(* Logix 5000 project; controller L3 vendor 1 type 14 code 92 rev 20.12; software revision 20.04; part 4 of 9 *)
(* tags used below, declared in another part *)
   B3 : DINT[100];
   L3_stat : DINT[20];
   N20 : DINT[200];
   N21 : DINT[200];
   N7 : DINT[200];
   N9 : DINT[200];   // niveau decapage vers lancy (n9[10) ;;N9[70]
   NCOM : INT[20];
   new_def_decap : BOOL;
   s_def_new : DINT;
   s_def_old : DINT;
   stat_L3 : DINT[20];
   T4 : TIMER[180];
(* _2_GENERAL, continued *)

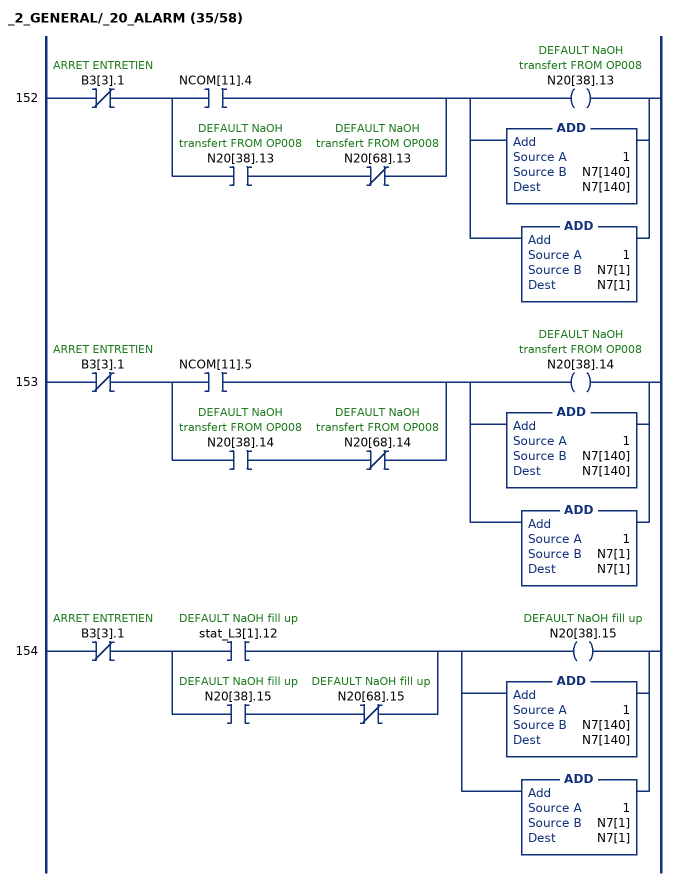
   [picture p50: _2_GENERAL/_20_ALARM rungs 152-154]
   152: XIO(B3[3].1)[XIC(NCOM[11].4) ,XIC(N20[38].13) XIO(N20[68].13) ][OTE(N20[38].13) ,ADD(1,N7[140],N7[140]) ,ADD(1,N7[1],N7[1]) ];
   153: XIO(B3[3].1)[XIC(NCOM[11].5) ,XIC(N20[38].14) XIO(N20[68].14) ][OTE(N20[38].14) ,ADD(1,N7[140],N7[140]) ,ADD(1,N7[1],N7[1]) ];
   154: XIO(B3[3].1)[XIC(stat_L3[1].12) ,XIC(N20[38].15) XIO(N20[68].15) ][OTE(N20[38].15) ,ADD(1,N7[140],N7[140]) ,ADD(1,N7[1],N7[1]) ];
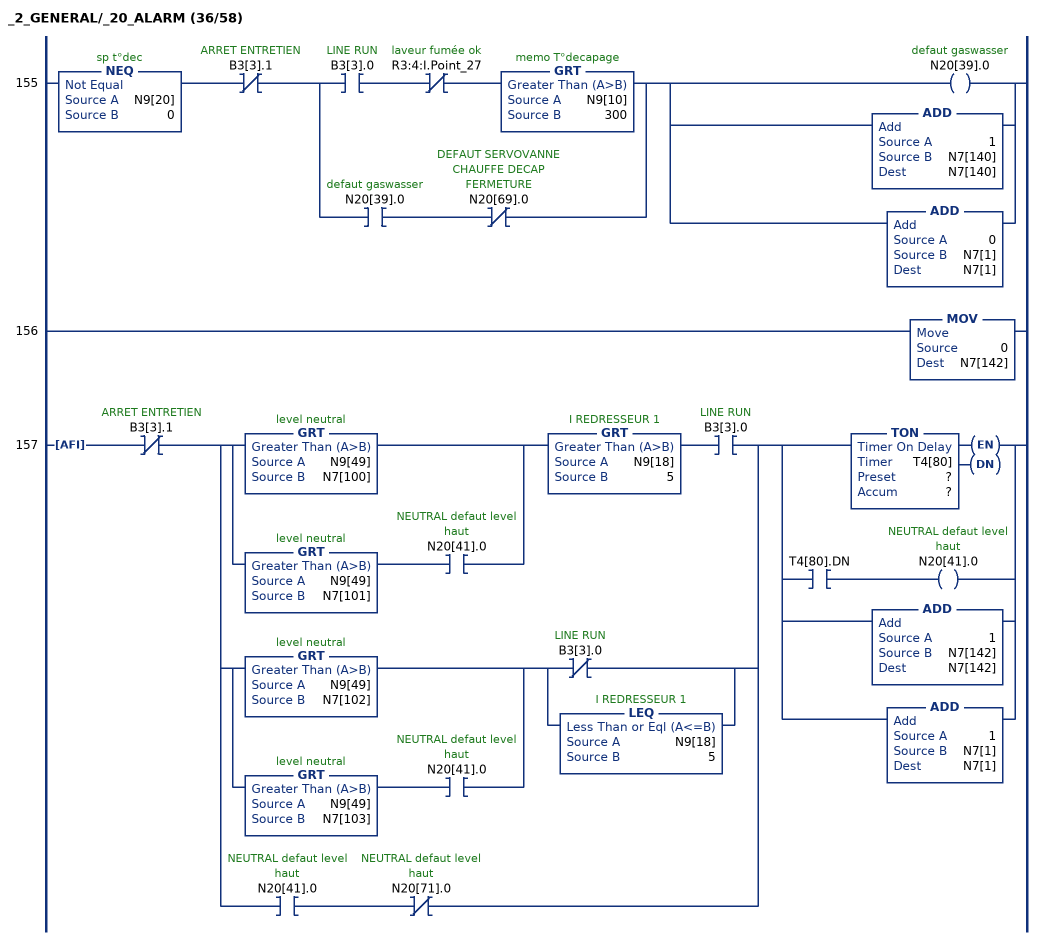
   155: NEQ(N9[20],0)XIO(B3[3].1)[XIC(B3[3].0) XIO(R3:4:I.Point_27) GRT(N9[10],300) ,XIC(N20[39].0) XIO(N20[69].0) ][OTE(N20[39].0) ,ADD(1,N7[140],N7[140]) ,ADD(0,N7[1],N7[1]) ];
   156: MOV(0,N7[142]);
   157: AFI()XIO(B3[3].1)[[GRT(N9[49],N7[100]) ,GRT(N9[49],N7[101]) XIC(N20[41].0) ] GRT(N9[18],5) XIC(B3[3].0) ,[GRT(N9[49],N7[102]) ,GRT(N9[49],N7[103]) XIC(N20[41].0) ] [XIO(B3[3].0) ,LEQ(N9[18],5) ] ,XIC(N20[41].0) XIO(N20[71].0) ][TON(T4[80],?,?) ,XIC(T4[80].DN) OTE(N20[41].0) ,ADD(1,N7[142],N7[142]) ,ADD(1,N7[1],N7[1]) ];
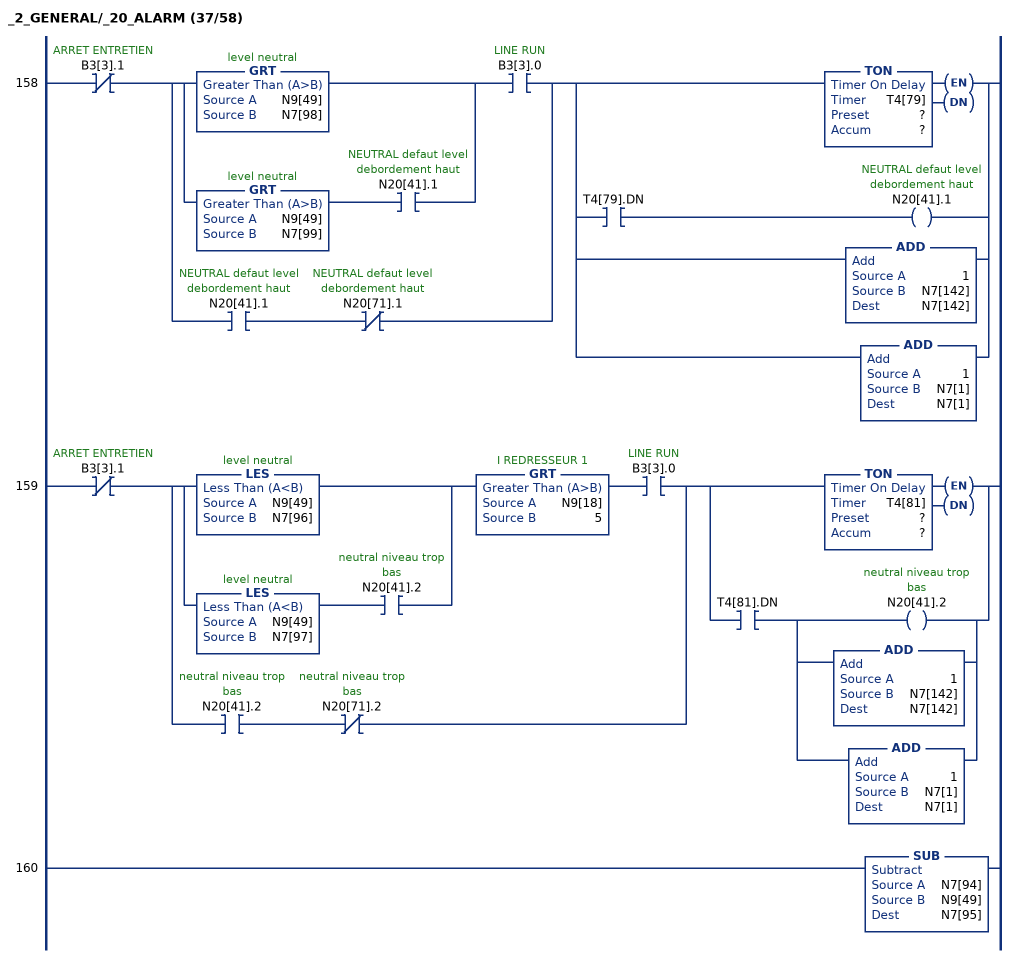
   158: XIO(B3[3].1)[[GRT(N9[49],N7[98]) ,GRT(N9[49],N7[99]) XIC(N20[41].1) ] XIC(B3[3].0) ,XIC(N20[41].1) XIO(N20[71].1) ][TON(T4[79],?,?) ,XIC(T4[79].DN) OTE(N20[41].1) ,ADD(1,N7[142],N7[142]) ,ADD(1,N7[1],N7[1]) ];
   159: XIO(B3[3].1)[[LES(N9[49],N7[96]) ,LES(N9[49],N7[97]) XIC(N20[41].2) ] GRT(N9[18],5) XIC(B3[3].0) ,XIC(N20[41].2) XIO(N20[71].2) ][TON(T4[81],?,?) ,XIC(T4[81].DN) [OTE(N20[41].2) ,ADD(1,N7[142],N7[142]) ,ADD(1,N7[1],N7[1]) ] ];
   160: SUB(N7[94],N9[49],N7[95]);
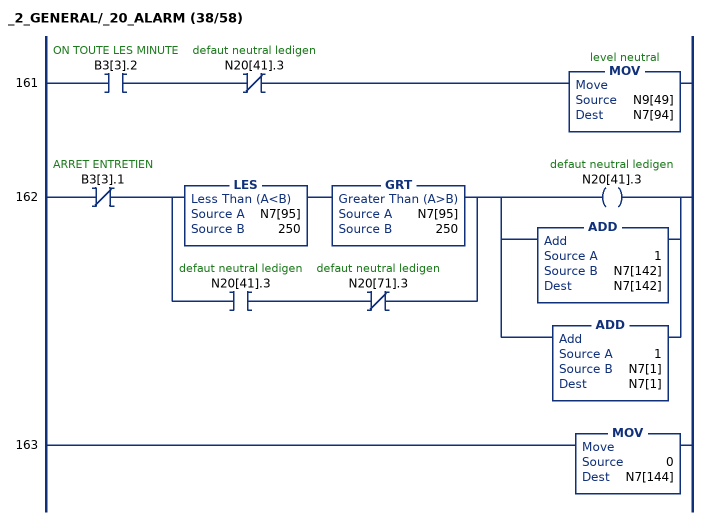
   161: XIC(B3[3].2)XIO(N20[41].3)MOV(N9[49],N7[94]);
   162: XIO(B3[3].1)[LES(N7[95],250) GRT(N7[95],250) ,XIC(N20[41].3) XIO(N20[71].3) ][OTE(N20[41].3) ,ADD(1,N7[142],N7[142]) ,ADD(1,N7[1],N7[1]) ];
   163: MOV(0,N7[144]);
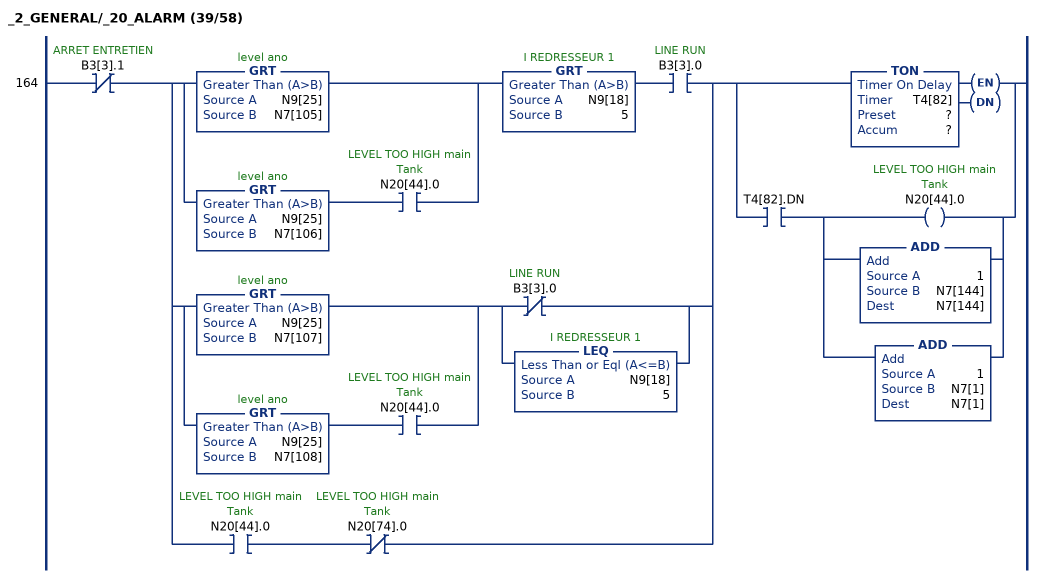
   164: XIO(B3[3].1)[[GRT(N9[25],N7[105]) ,GRT(N9[25],N7[106]) XIC(N20[44].0) ] GRT(N9[18],5) XIC(B3[3].0) ,[GRT(N9[25],N7[107]) ,GRT(N9[25],N7[108]) XIC(N20[44].0) ] [XIO(B3[3].0) ,LEQ(N9[18],5) ] ,XIC(N20[44].0) XIO(N20[74].0) ][TON(T4[82],?,?) ,XIC(T4[82].DN) [OTE(N20[44].0) ,ADD(1,N7[144],N7[144]) ,ADD(1,N7[1],N7[1]) ] ];
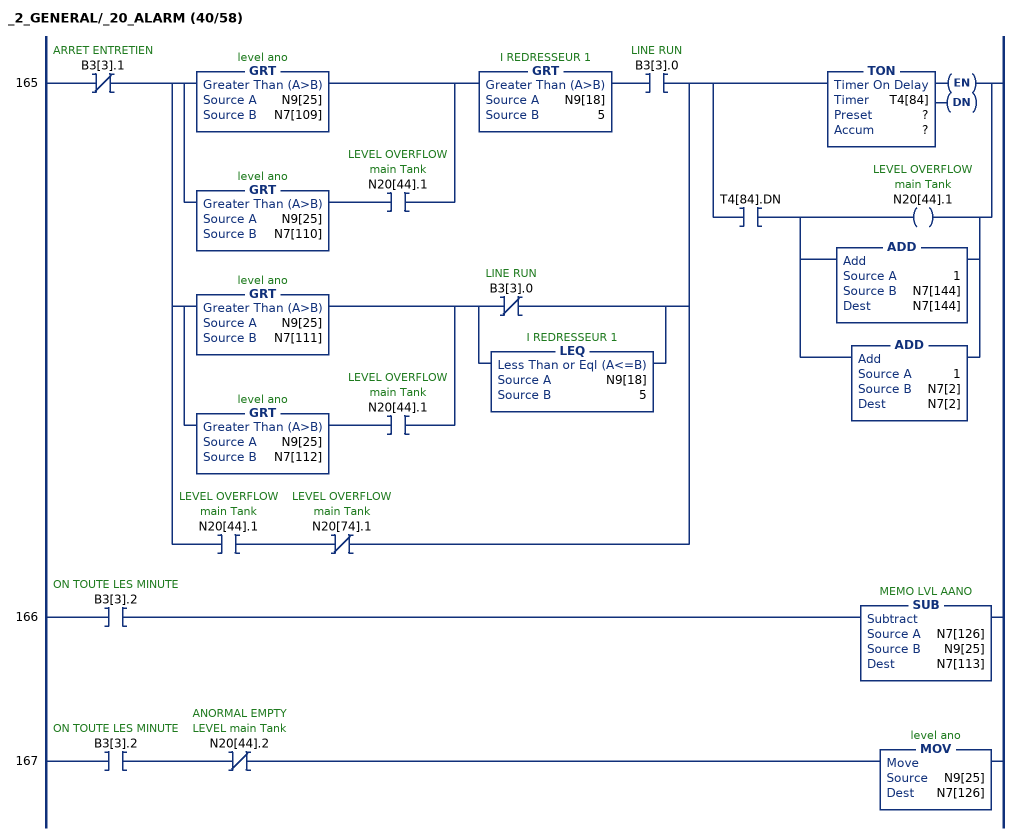
   165: XIO(B3[3].1)[[GRT(N9[25],N7[109]) ,GRT(N9[25],N7[110]) XIC(N20[44].1) ] GRT(N9[18],5) XIC(B3[3].0) ,[GRT(N9[25],N7[111]) ,GRT(N9[25],N7[112]) XIC(N20[44].1) ] [XIO(B3[3].0) ,LEQ(N9[18],5) ] ,XIC(N20[44].1) XIO(N20[74].1) ][TON(T4[84],?,?) ,XIC(T4[84].DN) [OTE(N20[44].1) ,ADD(1,N7[144],N7[144]) ,ADD(1,N7[2],N7[2]) ] ];
   166: XIC(B3[3].2)SUB(N7[126],N9[25],N7[113]);
   167: XIC(B3[3].2)XIO(N20[44].2)MOV(N9[25],N7[126]);
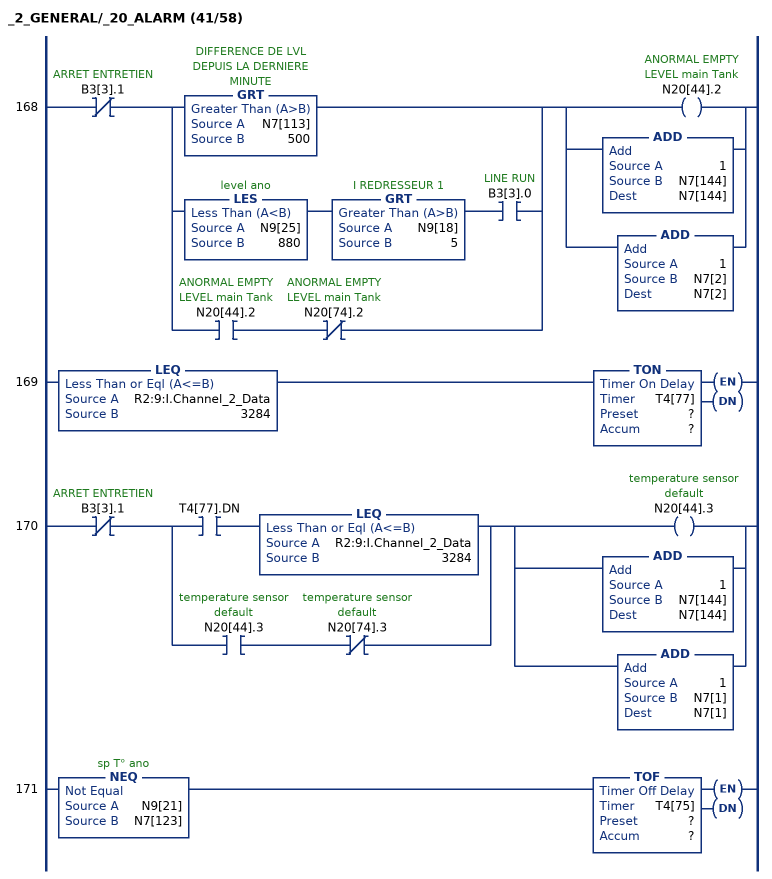
   168: XIO(B3[3].1)[GRT(N7[113],500) ,LES(N9[25],880) GRT(N9[18],5) XIC(B3[3].0) ,XIC(N20[44].2) XIO(N20[74].2) ][OTE(N20[44].2) ,ADD(1,N7[144],N7[144]) ,ADD(1,N7[2],N7[2]) ];
   169: LEQ(R2:9:I.Channel_2_Data,3284)TON(T4[77],?,?);
   170: XIO(B3[3].1)[XIC(T4[77].DN) LEQ(R2:9:I.Channel_2_Data,3284) ,XIC(N20[44].3) XIO(N20[74].3) ][OTE(N20[44].3) ,ADD(1,N7[144],N7[144]) ,ADD(1,N7[1],N7[1]) ];
   171: NEQ(N9[21],N7[123])TOF(T4[75],?,?);
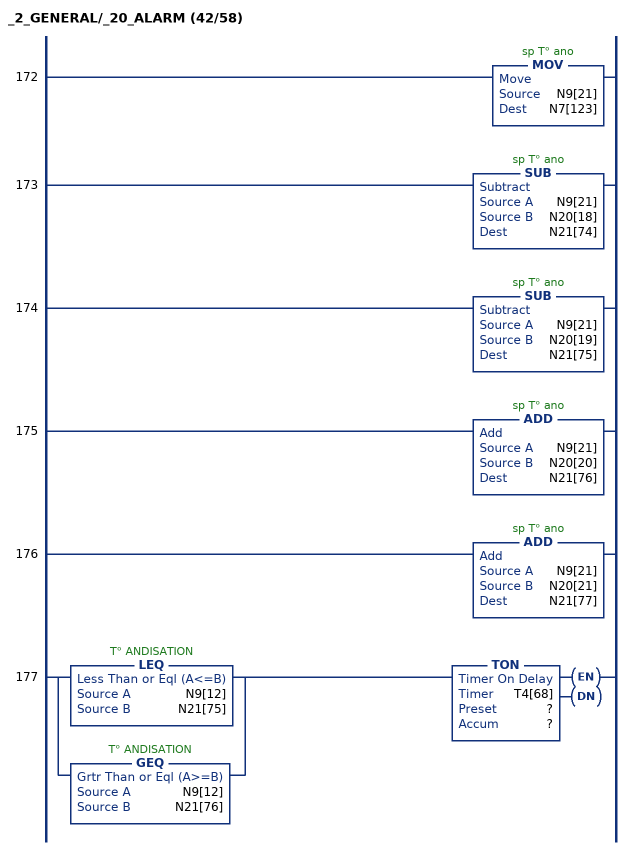
   172: MOV(N9[21],N7[123]);
   173: SUB(N9[21],N20[18],N21[74]);
   174: SUB(N9[21],N20[19],N21[75]);
   175: ADD(N9[21],N20[20],N21[76]);
   176: ADD(N9[21],N20[21],N21[77]);
   177: [LEQ(N9[12],N21[75]) ,GEQ(N9[12],N21[76]) ]TON(T4[68],?,?);
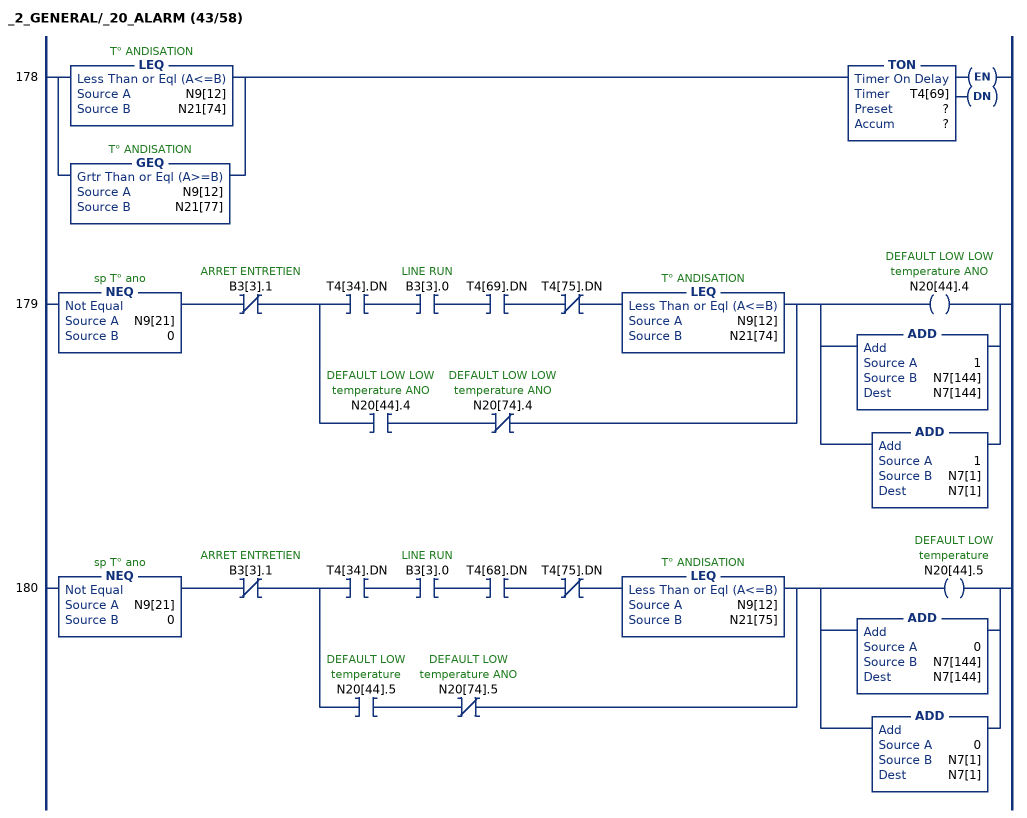
   178: [LEQ(N9[12],N21[74]) ,GEQ(N9[12],N21[77]) ]TON(T4[69],?,?);
   179: NEQ(N9[21],0)XIO(B3[3].1)[XIC(T4[34].DN) XIC(B3[3].0) XIC(T4[69].DN) XIO(T4[75].DN) LEQ(N9[12],N21[74]) ,XIC(N20[44].4) XIO(N20[74].4) ][OTE(N20[44].4) ,ADD(1,N7[144],N7[144]) ,ADD(1,N7[1],N7[1]) ];
   180: NEQ(N9[21],0)XIO(B3[3].1)[XIC(T4[34].DN) XIC(B3[3].0) XIC(T4[68].DN) XIO(T4[75].DN) LEQ(N9[12],N21[75]) ,XIC(N20[44].5) XIO(N20[74].5) ][OTE(N20[44].5) ,ADD(0,N7[144],N7[144]) ,ADD(0,N7[1],N7[1]) ];
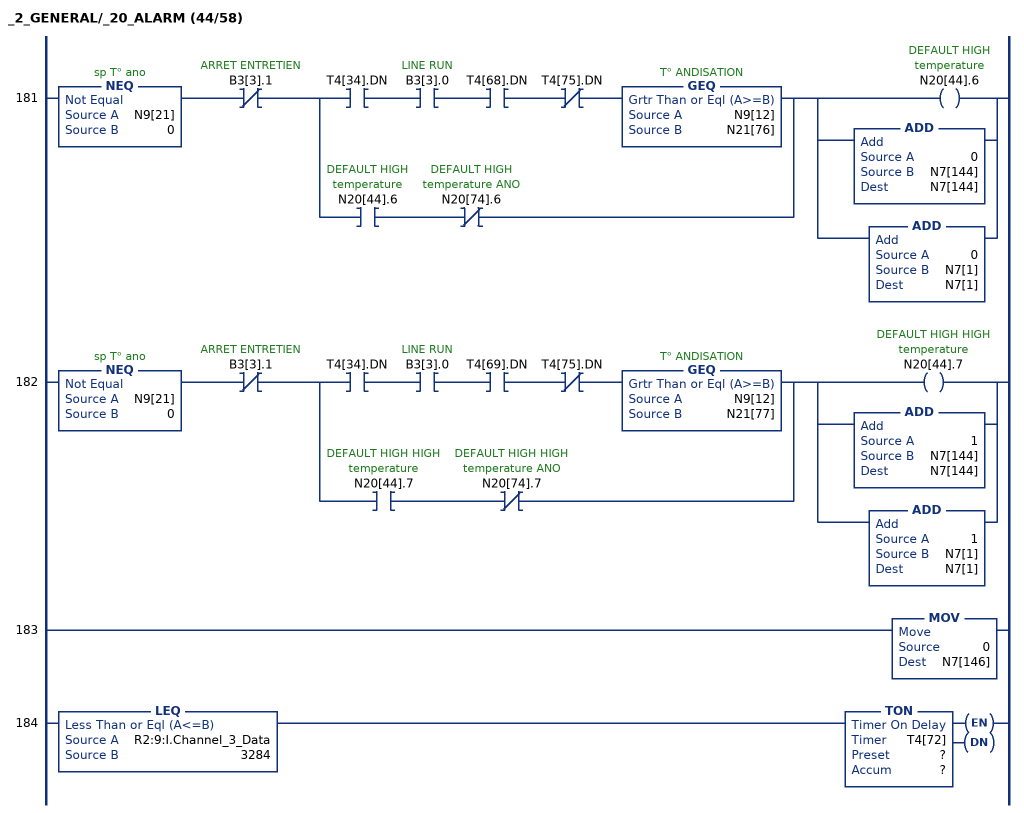
   181: NEQ(N9[21],0)XIO(B3[3].1)[XIC(T4[34].DN) XIC(B3[3].0) XIC(T4[68].DN) XIO(T4[75].DN) GEQ(N9[12],N21[76]) ,XIC(N20[44].6) XIO(N20[74].6) ][OTE(N20[44].6) ,ADD(0,N7[144],N7[144]) ,ADD(0,N7[1],N7[1]) ];
   182: NEQ(N9[21],0)XIO(B3[3].1)[XIC(T4[34].DN) XIC(B3[3].0) XIC(T4[69].DN) XIO(T4[75].DN) GEQ(N9[12],N21[77]) ,XIC(N20[44].7) XIO(N20[74].7) ][OTE(N20[44].7) ,ADD(1,N7[144],N7[144]) ,ADD(1,N7[1],N7[1]) ];
   183: MOV(0,N7[146]);
   184: LEQ(R2:9:I.Channel_3_Data,3284)TON(T4[72],?,?);
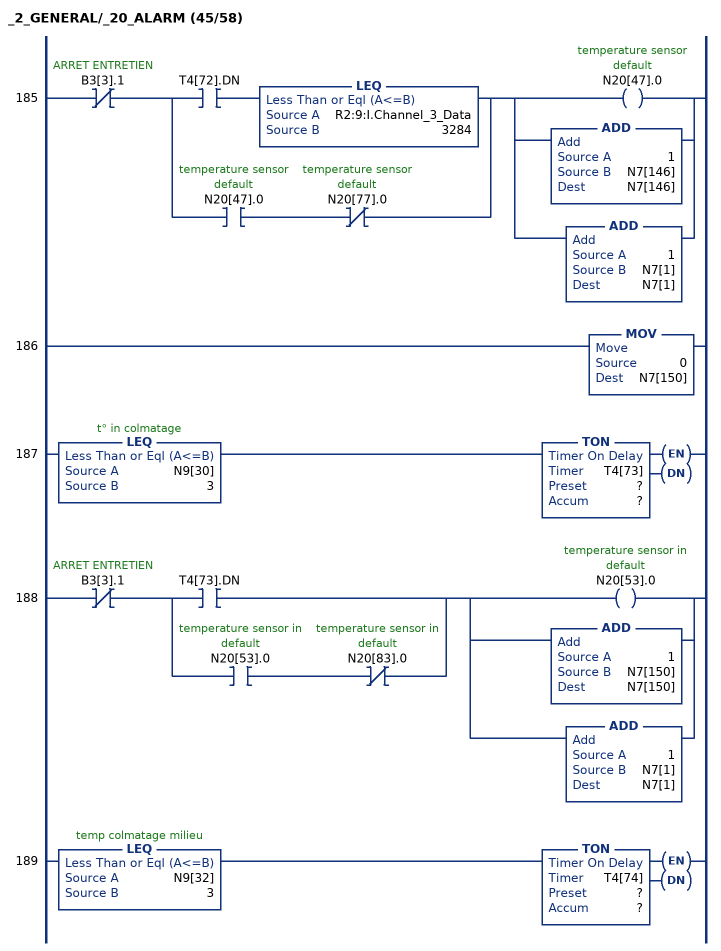
   185: XIO(B3[3].1)[XIC(T4[72].DN) LEQ(R2:9:I.Channel_3_Data,3284) ,XIC(N20[47].0) XIO(N20[77].0) ][OTE(N20[47].0) ,ADD(1,N7[146],N7[146]) ,ADD(1,N7[1],N7[1]) ];
   186: MOV(0,N7[150]);
   187: LEQ(N9[30],3)TON(T4[73],?,?);
   188: XIO(B3[3].1)[XIC(T4[73].DN) ,XIC(N20[53].0) XIO(N20[83].0) ][OTE(N20[53].0) ,ADD(1,N7[150],N7[150]) ,ADD(1,N7[1],N7[1]) ];
   189: LEQ(N9[32],3)TON(T4[74],?,?);
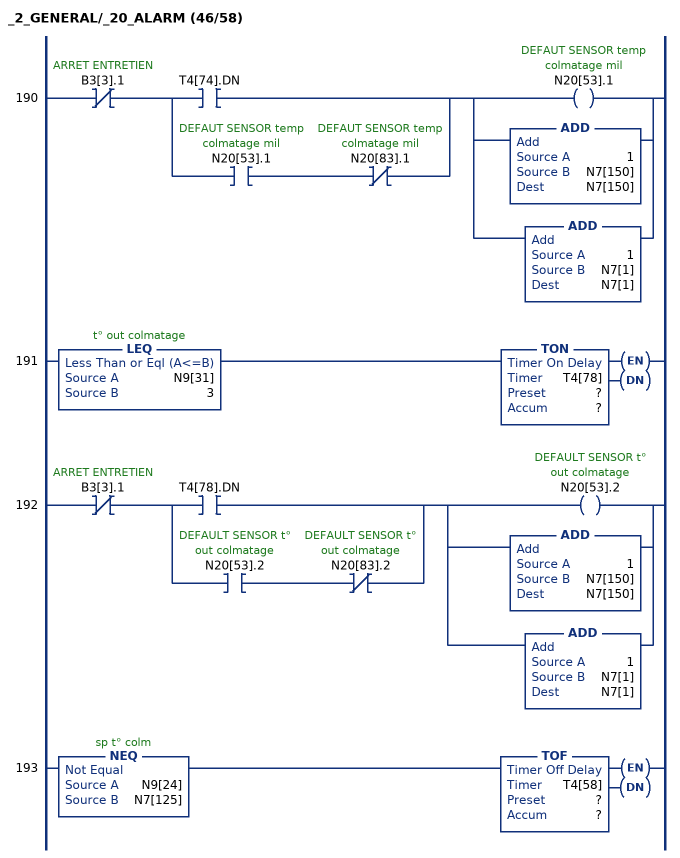
   190: XIO(B3[3].1)[XIC(T4[74].DN) ,XIC(N20[53].1) XIO(N20[83].1) ][OTE(N20[53].1) ,ADD(1,N7[150],N7[150]) ,ADD(1,N7[1],N7[1]) ];
   191: LEQ(N9[31],3)TON(T4[78],?,?);
   192: XIO(B3[3].1)[XIC(T4[78].DN) ,XIC(N20[53].2) XIO(N20[83].2) ][OTE(N20[53].2) ,ADD(1,N7[150],N7[150]) ,ADD(1,N7[1],N7[1]) ];
   193: NEQ(N9[24],N7[125])TOF(T4[58],?,?);
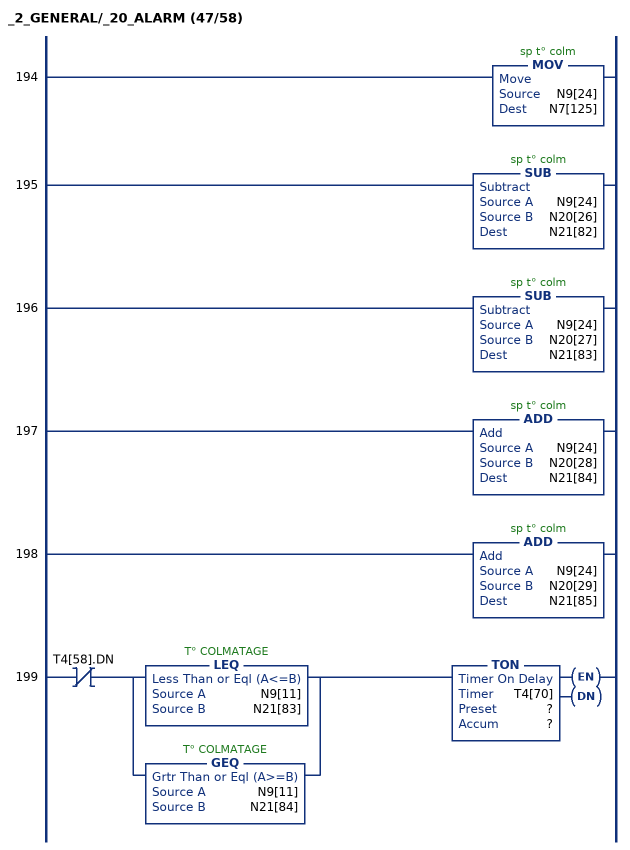
   194: MOV(N9[24],N7[125]);
   195: SUB(N9[24],N20[26],N21[82]);
   196: SUB(N9[24],N20[27],N21[83]);
   197: ADD(N9[24],N20[28],N21[84]);
   198: ADD(N9[24],N20[29],N21[85]);
   199: XIO(T4[58].DN)[LEQ(N9[11],N21[83]) ,GEQ(N9[11],N21[84]) ]TON(T4[70],?,?);
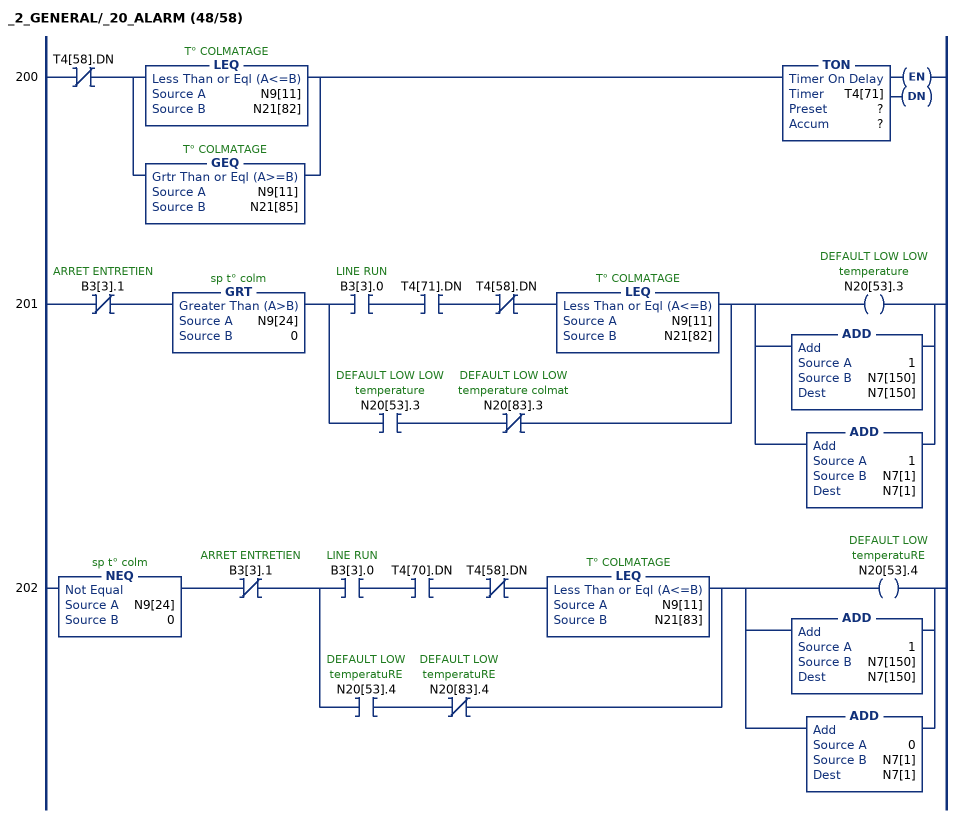
   200: XIO(T4[58].DN)[LEQ(N9[11],N21[82]) ,GEQ(N9[11],N21[85]) ]TON(T4[71],?,?);
   201: XIO(B3[3].1)GRT(N9[24],0)[XIC(B3[3].0) XIC(T4[71].DN) XIO(T4[58].DN) LEQ(N9[11],N21[82]) ,XIC(N20[53].3) XIO(N20[83].3) ][OTE(N20[53].3) ,ADD(1,N7[150],N7[150]) ,ADD(1,N7[1],N7[1]) ];
   202: NEQ(N9[24],0)XIO(B3[3].1)[XIC(B3[3].0) XIC(T4[70].DN) XIO(T4[58].DN) LEQ(N9[11],N21[83]) ,XIC(N20[53].4) XIO(N20[83].4) ][OTE(N20[53].4) ,ADD(1,N7[150],N7[150]) ,ADD(0,N7[1],N7[1]) ];
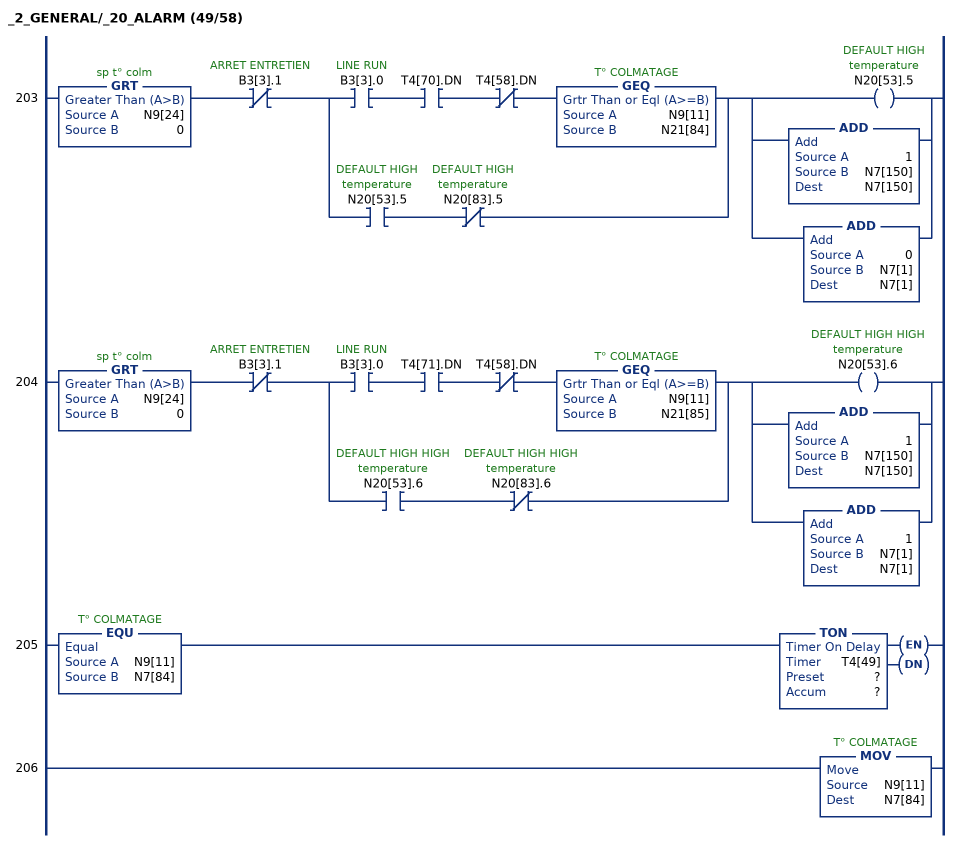
   203: GRT(N9[24],0)XIO(B3[3].1)[XIC(B3[3].0) XIC(T4[70].DN) XIO(T4[58].DN) GEQ(N9[11],N21[84]) ,XIC(N20[53].5) XIO(N20[83].5) ][OTE(N20[53].5) ,ADD(1,N7[150],N7[150]) ,ADD(0,N7[1],N7[1]) ];
   204: GRT(N9[24],0)XIO(B3[3].1)[XIC(B3[3].0) XIC(T4[71].DN) XIO(T4[58].DN) GEQ(N9[11],N21[85]) ,XIC(N20[53].6) XIO(N20[83].6) ][OTE(N20[53].6) ,ADD(1,N7[150],N7[150]) ,ADD(1,N7[1],N7[1]) ];
   205: EQU(N9[11],N7[84])TON(T4[49],?,?);
   206: MOV(N9[11],N7[84]);
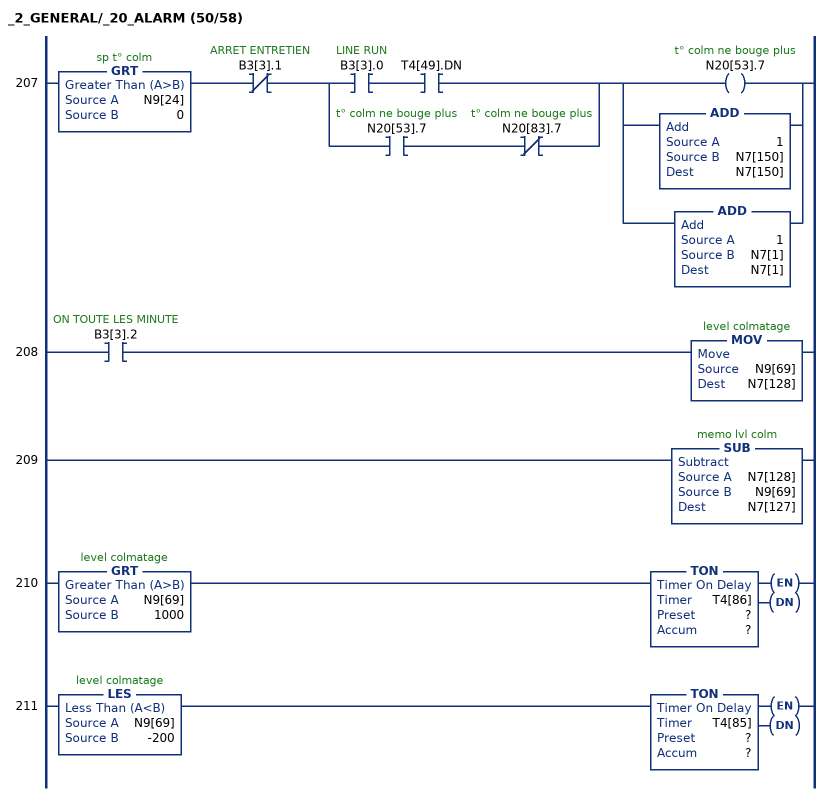
   207: GRT(N9[24],0)XIO(B3[3].1)[XIC(B3[3].0) XIC(T4[49].DN) ,XIC(N20[53].7) XIO(N20[83].7) ][OTE(N20[53].7) ,ADD(1,N7[150],N7[150]) ,ADD(1,N7[1],N7[1]) ];
   208: XIC(B3[3].2)MOV(N9[69],N7[128]);
   209: SUB(N7[128],N9[69],N7[127]);
   210: GRT(N9[69],1000)TON(T4[86],?,?);
   211: LES(N9[69],-200)TON(T4[85],?,?);
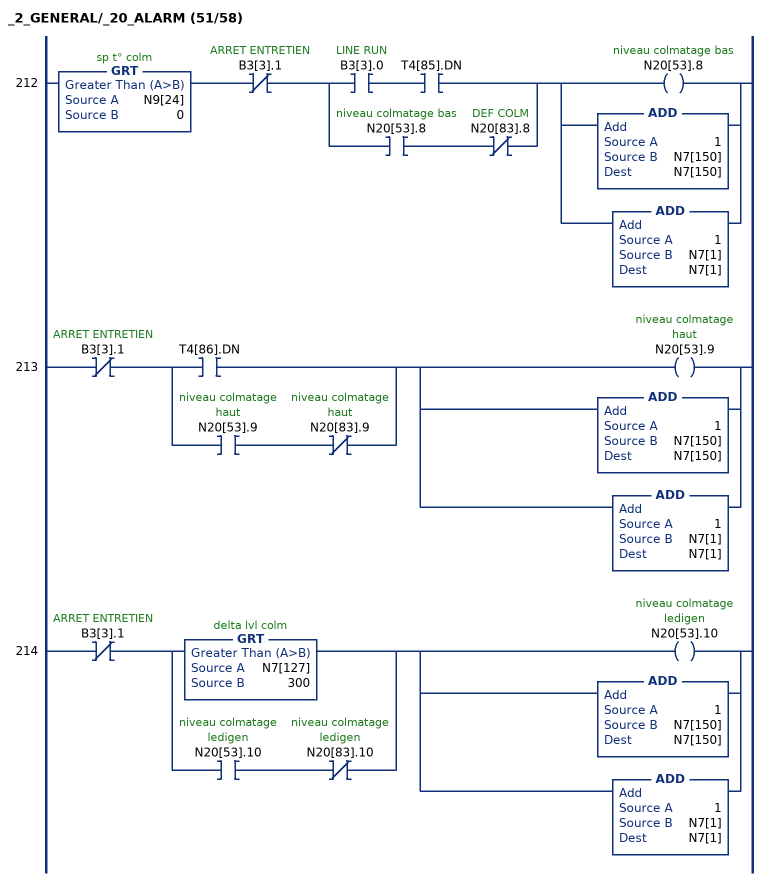
   212: GRT(N9[24],0)XIO(B3[3].1)[XIC(B3[3].0) XIC(T4[85].DN) ,XIC(N20[53].8) XIO(N20[83].8) ][OTE(N20[53].8) ,ADD(1,N7[150],N7[150]) ,ADD(1,N7[1],N7[1]) ];
   213: XIO(B3[3].1)[XIC(T4[86].DN) ,XIC(N20[53].9) XIO(N20[83].9) ][OTE(N20[53].9) ,ADD(1,N7[150],N7[150]) ,ADD(1,N7[1],N7[1]) ];
   214: XIO(B3[3].1)[GRT(N7[127],300) ,XIC(N20[53].10) XIO(N20[83].10) ][OTE(N20[53].10) ,ADD(1,N7[150],N7[150]) ,ADD(1,N7[1],N7[1]) ];
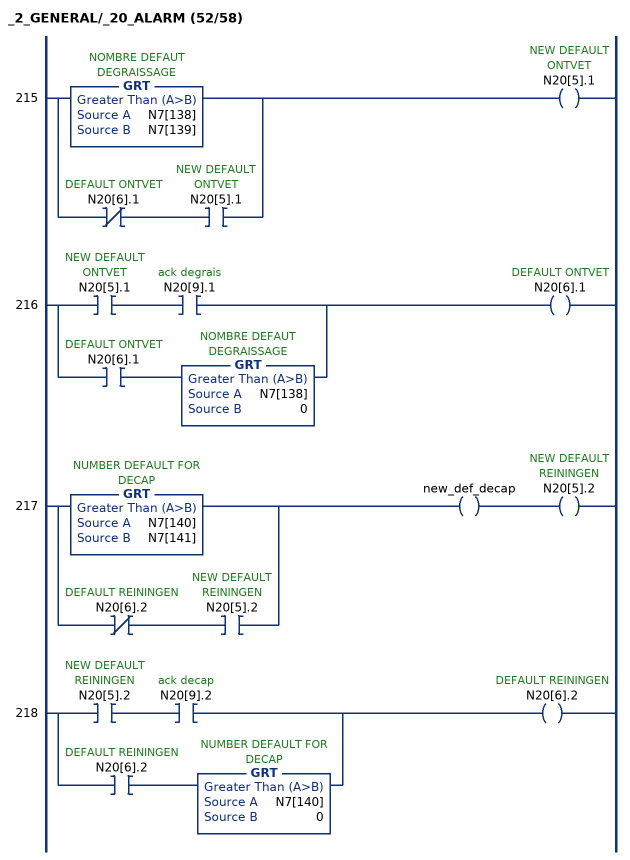
   215: [GRT(N7[138],N7[139]) ,XIO(N20[6].1) XIC(N20[5].1) ]OTE(N20[5].1);
   216: [XIC(N20[5].1) XIC(N20[9].1) ,XIC(N20[6].1) GRT(N7[138],0) ]OTE(N20[6].1);
   217: [GRT(N7[140],N7[141]) ,XIO(N20[6].2) XIC(N20[5].2) ]OTE(new_def_decap)OTE(N20[5].2);
   218: [XIC(N20[5].2) XIC(N20[9].2) ,XIC(N20[6].2) GRT(N7[140],0) ]OTE(N20[6].2);
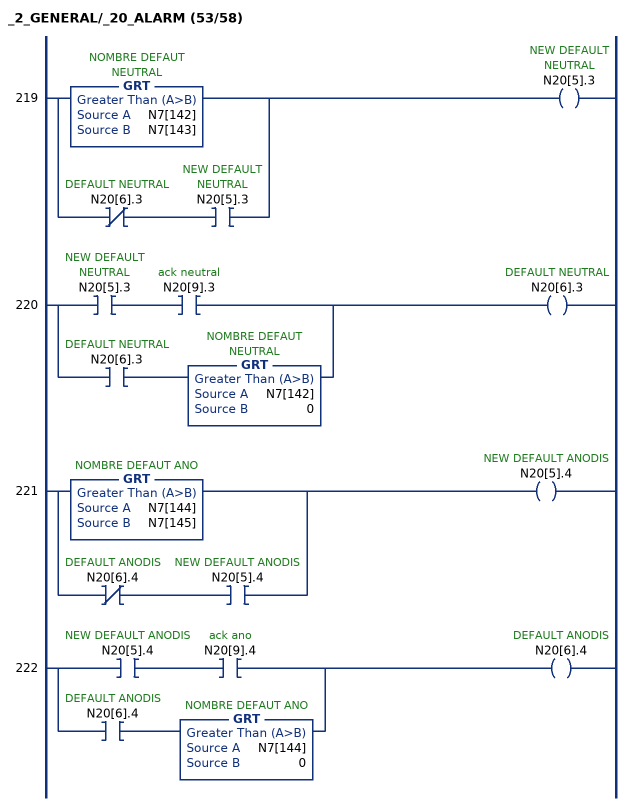
   219: [GRT(N7[142],N7[143]) ,XIO(N20[6].3) XIC(N20[5].3) ]OTE(N20[5].3);
   220: [XIC(N20[5].3) XIC(N20[9].3) ,XIC(N20[6].3) GRT(N7[142],0) ]OTE(N20[6].3);
   221: [GRT(N7[144],N7[145]) ,XIO(N20[6].4) XIC(N20[5].4) ]OTE(N20[5].4);
   222: [XIC(N20[5].4) XIC(N20[9].4) ,XIC(N20[6].4) GRT(N7[144],0) ]OTE(N20[6].4);
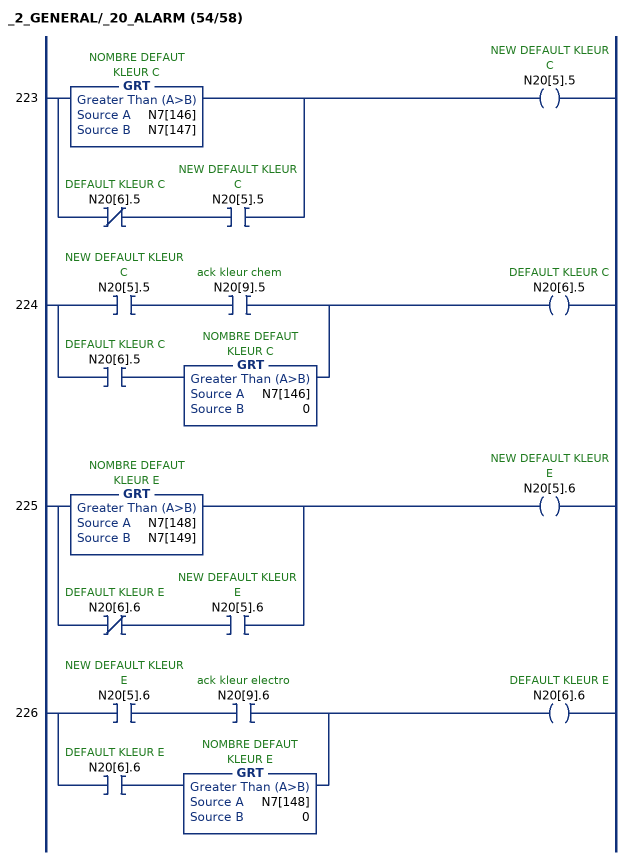
   223: [GRT(N7[146],N7[147]) ,XIO(N20[6].5) XIC(N20[5].5) ]OTE(N20[5].5);
   224: [XIC(N20[5].5) XIC(N20[9].5) ,XIC(N20[6].5) GRT(N7[146],0) ]OTE(N20[6].5);
   225: [GRT(N7[148],N7[149]) ,XIO(N20[6].6) XIC(N20[5].6) ]OTE(N20[5].6);
   226: [XIC(N20[5].6) XIC(N20[9].6) ,XIC(N20[6].6) GRT(N7[148],0) ]OTE(N20[6].6);
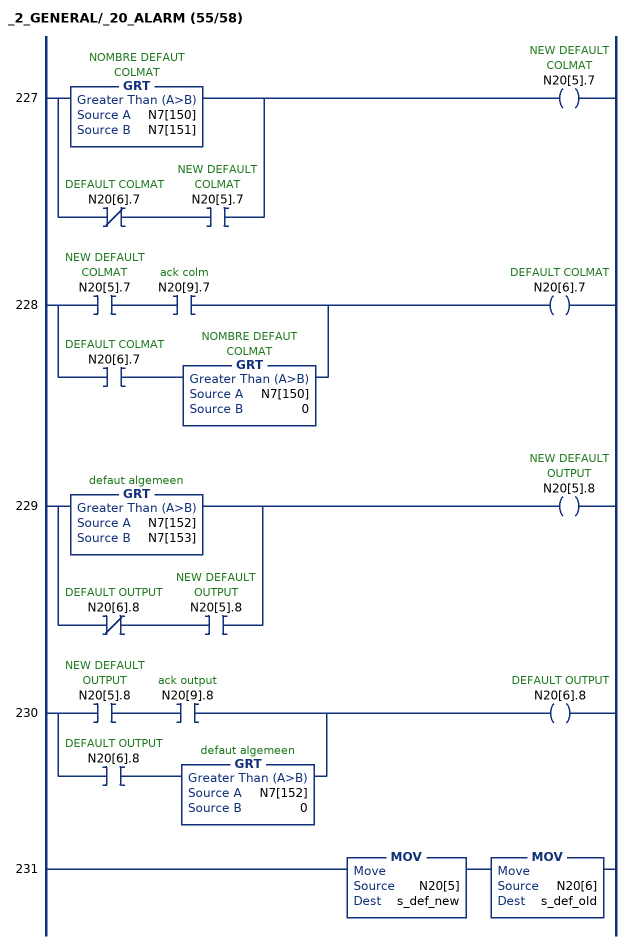
   227: [GRT(N7[150],N7[151]) ,XIO(N20[6].7) XIC(N20[5].7) ]OTE(N20[5].7);
   228: [XIC(N20[5].7) XIC(N20[9].7) ,XIC(N20[6].7) GRT(N7[150],0) ]OTE(N20[6].7);
   229: [GRT(N7[152],N7[153]) ,XIO(N20[6].8) XIC(N20[5].8) ]OTE(N20[5].8);
   230: [XIC(N20[5].8) XIC(N20[9].8) ,XIC(N20[6].8) GRT(N7[152],0) ]OTE(N20[6].8);
   231: MOV(N20[5],s_def_new)MOV(N20[6],s_def_old);
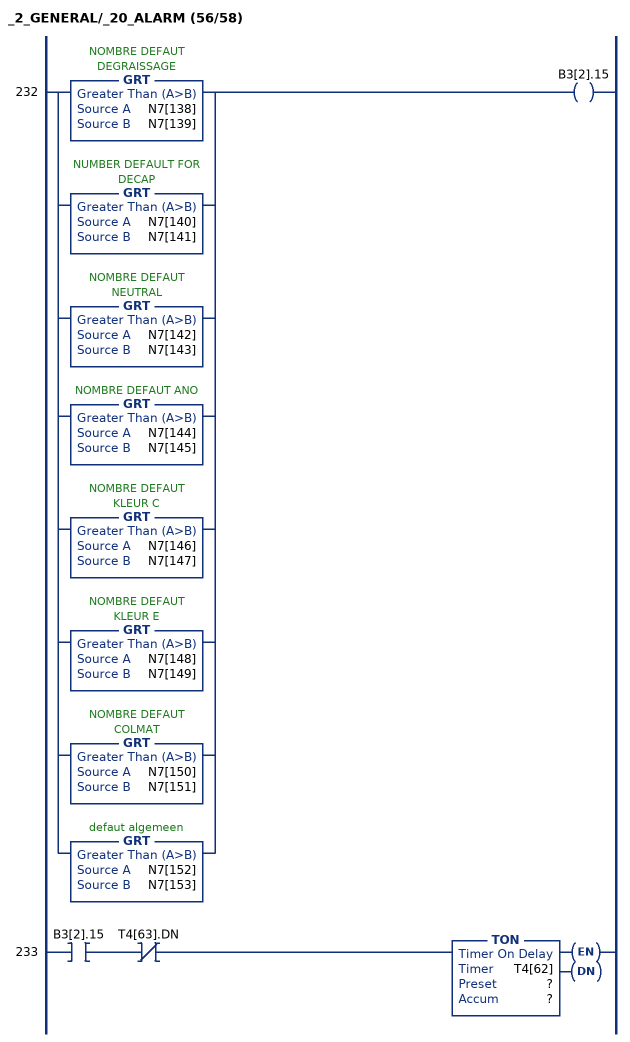
   232: [GRT(N7[138],N7[139]) ,GRT(N7[140],N7[141]) ,GRT(N7[142],N7[143]) ,GRT(N7[144],N7[145]) ,GRT(N7[146],N7[147]) ,GRT(N7[148],N7[149]) ,GRT(N7[150],N7[151]) ,GRT(N7[152],N7[153]) ]OTE(B3[2].15);
   233: XIC(B3[2].15)XIO(T4[63].DN)TON(T4[62],?,?);
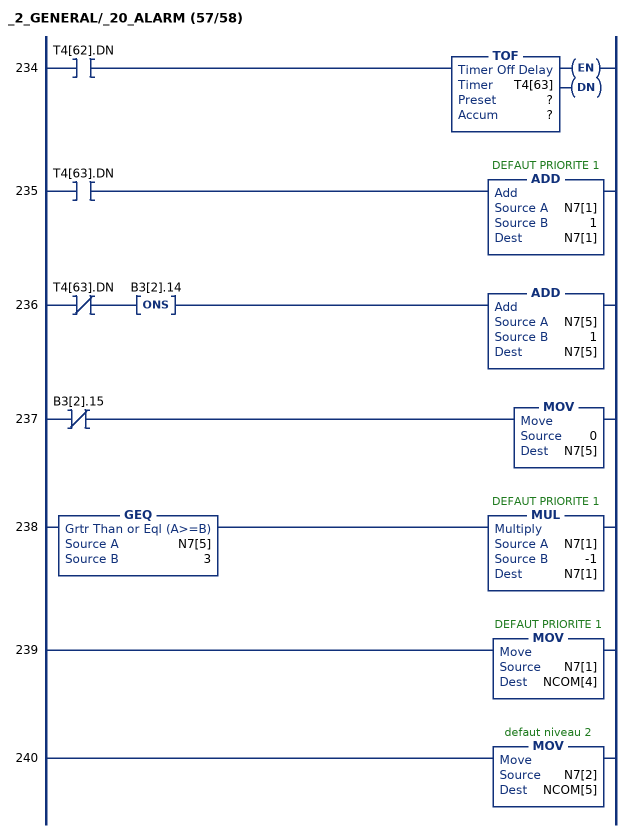
   234: XIC(T4[62].DN)TOF(T4[63],?,?);
   235: XIC(T4[63].DN)ADD(N7[1],1,N7[1]);
   236: XIO(T4[63].DN)ONS(B3[2].14)ADD(N7[5],1,N7[5]);
   237: XIO(B3[2].15)MOV(0,N7[5]);
   238: GEQ(N7[5],3)MUL(N7[1],-1,N7[1]);
   239: MOV(N7[1],NCOM[4]);
   240: MOV(N7[2],NCOM[5]);
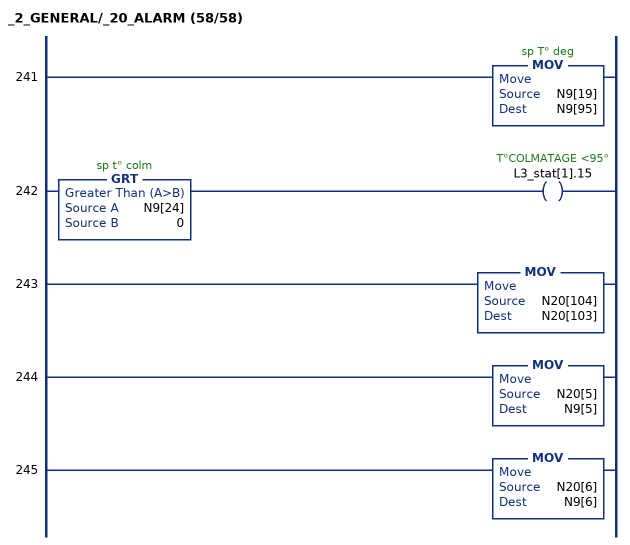
   241: MOV(N9[19],N9[95]);
   242: GRT(N9[24],0)OTE(L3_stat[1].15);
   243: MOV(N20[104],N20[103]);
   244: MOV(N20[5],N9[5]);
   245: MOV(N20[6],N9[6]);
END_ROUTINE
